FUNCTION_BLOCK INTERNAL FB_AlarmActionBuilder IMPLEMENTS I_AlarmActionBy, I_AlarmActions
VAR
	_alarmAction 	: (ACTION_ACKNOWLEDGE, ACTTION_RAISE, ACTION_DEACTIVATE);
	_selectedAlarm	: REFERENCE TO ST_AlarmInfo;
	_alarmManager	: REFERENCE TO FB_AlarmManager;
END_VAR

VAR CONSTANT
	_emptyAlarm		: ST_AlarmInfo;	
END_VAR

METHOD Acknowledge : I_AlarmActionBy
VAR_INPUT
END_VAR
_alarmAction := ACTION_ACKNOWLEDGE;
Acknowledge := THIS^;
END_METHOD

// Executes the action by looking for the alarm with the provided ID
METHOD ById
VAR_INPUT
	Id	: T_ArrayIndexer;
END_VAR
VAR
	i	: T_ArrayIndexer;
END_VAR
IF NOT __ISVALIDREF(_alarmManager.GetAlarmById(Id)) THEN
	RETURN;
END_IF

_selectedAlarm REF= _alarmManager.GetAlarmById(Id);
DoAction();
END_METHOD

// Executes the action by looking for the alarm with the provided name
METHOD ByName
VAR_INPUT
	name	: Tc2_System.T_MaxString;
END_VAR

VAR_INST
	i	: T_ArrayIndexer;
END_VAR
IF NOT __ISVALIDREF(_alarmManager.GetAlarmByName(name)) THEN
	RETURN;
END_IF
_selectedAlarm REF= _alarmManager.GetAlarmByName(name);
DoAction();
END_METHOD

METHOD Deactivate : I_AlarmActionBy
VAR_INPUT
END_VAR
_alarmAction := ACTION_DEACTIVATE;
Deactivate := THIS^;
END_METHOD

METHOD PRIVATE DoAction
CASE _alarmAction OF
	ACTION_ACKNOWLEDGE:
		_alarmManager.AcknowledgeAlarm(_selectedAlarm);
	ACTTION_RAISE:
		_alarmManager.RaiseAlarm(_selectedAlarm);
	ACTION_DEACTIVATE:
		_alarmManager.DeactivateAlarm(_selectedAlarm);
END_CASE
END_METHOD

METHOD FB_init : BOOL
VAR_INPUT
	bInitRetains : BOOL; // if TRUE, the retain variables are initialized (warm start / cold start)
	bInCopyCode : BOOL;  // if TRUE, the instance afterwards gets moved into the copy code (online change)
	alarmManager	: REFERENCE TO FB_AlarmManager;
END_VAR
_alarmManager REF= alarmManager;
END_METHOD

METHOD Raise : I_AlarmActionBy
VAR_INPUT
END_VAR
_alarmAction := ACTTION_RAISE;
Raise := THIS^;
END_METHOD

PROPERTY SelectedAlarm : REFERENCE TO ST_AlarmInfo
GET
END_GET
END_PROPERTY

END_FUNCTION_BLOCK

(* stored: Version 1.1.0.1, ProductVersion 3.1.4024.14
   POU FB_AlarmActionBuilder: Id {cf92893f-c46c-0cad-3a1f-3e982e8ce72f}, SpecialFunc None
   Method Acknowledge: Id {ec3b6a2d-f8f4-080c-39cc-793e7b4fefaf}
   Method ById: Id {15bccc9e-311d-07d8-07f9-0b551d64ab1f}
   Method ByName: Id {6c000c08-a5b9-0289-097f-bd36cbfd51af}
   Method Deactivate: Id {bed0843b-36b5-034a-232f-b416d6d0b76a}
   Method DoAction: Id {74be2ef5-dc73-017b-0666-72826976b57c}
   Method FB_init: Id {4e5f7e03-115f-04e9-1e03-129289791e84}
   Method Raise: Id {3af8436e-f397-0704-2860-c8f26cdb4adb}
   Property SelectedAlarm: Id {1a689882-c53b-047d-1338-4cd1c5ea1074}
   Get Get: Id {9ab70128-2027-0ed8-2720-fcca32b6fab7} *)
